(* CoDeSys 2.3.9.50 project: 4B.pr6 *)
(* Libraries: STANDARD.LB6 5.6.98 12:03:02 *)

(* POU MAIN, LD *)
PROGRAM MAIN
VAR
	Start AT %IX0.0: BOOL;
	Stack AT %IX0.1: BOOL;
	C1: CTU;
	x AT %QX0.3: BOOL;
	Conveyer1 AT %QX0.0: BOOL;
	t1: TON;
	Conveyer2 AT %QX0.1: BOOL;

END_VAR
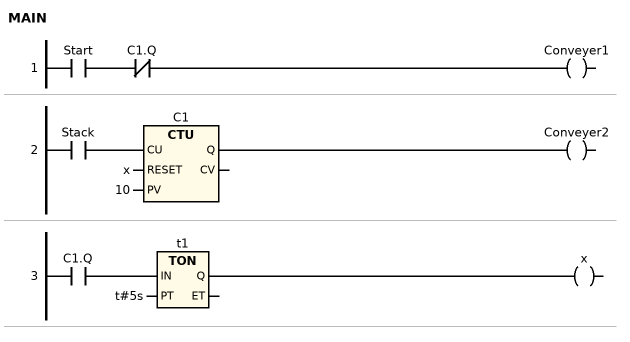
_LD_ (* Ladder Diagram *)
NETWORK 1
	[Start] - [/C1.Q] --- (Conveyer1)
NETWORK 2
	[Stack] - C1:CTU(CU: *, RESET: x, PV: 10) --- (Conveyer2)
NETWORK 3
	[C1.Q] - t1:TON(IN: *, PT: t#5s) --- (x)
_END_LD_
(* the same logic as Structured Text *)
(* Network 1 *)
Conveyer1 := Start AND NOT C1.Q;
(* Network 2 *)
C1(CU := Stack, RESET := x, PV := 10);
Conveyer2 := C1.Q;
(* Network 3 *)
t1(IN := C1.Q, PT := t#5s);
x := t1.Q;
END_PROGRAM
